(* PLC project PLC1, Beckhoff Automation GmbH TwinCAT PLC Control 3.5.21.20 *)
(* stored: creationDateTime 2026-02-22T16:42:22.4417689, modificationDateTime 2026-02-22T16:42:22.4417689 *)

(* 
    DUT: ST_BatchMetadata
    Description: Contains administrative information about the production order.
*)
TYPE ST_BatchMetadata :
STRUCT
    sOrderNumberSAP : STRING := '14963766'; 
    sFactory        : STRING := 'BJ04';     
    nDepartment     : DINT := 5541;         
    nWorkcenter     : DINT := 5349;         
    sEquipmentId    : STRING := '588555';         
END_STRUCT
END_TYPE
